PROGRAM RunGrindingWheel
VAR
END_VAR

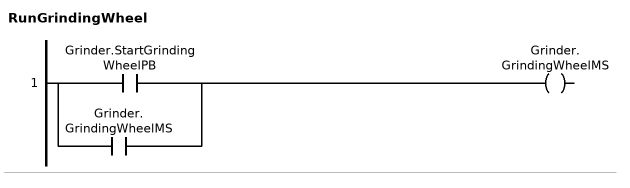
// NETWORK 1
Grinder.GrindingWheelMS := Grinder.StartGrindingWheelPB OR Grinder.GrindingWheelMS;

END_PROGRAM

(* stored: Version 1.1.0.1, ProductVersion 3.1.4024.6
   POU RunGrindingWheel: Id {3513ba1d-f760-4463-adfb-8672ce6298e9}, SpecialFunc None *)
